FUNCTION WORD_OF_DWORD : WORD
VAR_INPUT
	in : DWORD;
	N : BYTE;
END_VAR


(*
version 1.2	30. oct. 2008
programmer 	hugo
tested by	oscat

this function extracts a single word from the nth position from right (right is lowest byte)
the lower word (starting with Bit0 from in) is selected with N=0.
*)

WORD_OF_DWORD := DWORD_TO_WORD(SHR(in,SHL(n,4)));

(* revision history
hm	17. jan 2007	rev 1.0
	original version

hm	2. jan 2008		rev 1.1
	improved performance

hm	30. oct. 2008	rev 1.2
	improved performance
*)

END_FUNCTION

(* stored: Version 1.1.0.1, ProductVersion 3.1.4022.7
   POU WORD_OF_DWORD: Id {e4159dda-5fd9-4bf9-9d2f-990e74a0eb79}, SpecialFunc None *)
